KUKA KRL data list: FechaGarra.dat

&ACCESS RVO
&REL 1
&PARAM EDITMASK = *
DEFDAT FechaGarra

ENDDAT
